// Annex I I.8 - a bounded generated or taught route.
TYPE ST_RobotPointList :
STRUCT
    Points : ARRAY[1..PL_RobotPlanner.MAX_ROUTE_POINTS] OF ST_RobotPoint;
    Count  : INT;
END_STRUCT
END_TYPE

(* stored: Version 1.1.0.1, ProductVersion 3.1.4024.12
   DUT ST_RobotPointList: Id {5330e37c-aacd-4b94-9c92-b07c79b1689c} *)
